{attribute addProperty Name "Pneumatic cyclinder"}
FUNCTION_BLOCK fbPiston EXTENDS TcoCore.TcoComponent IMPLEMENTS IPistonGripper, IPistonHorizontal, IPistonVertical
VAR_INPUT
	iHomePositionSensor : BOOL;
	iWorkPositionSensor : BOOL;	
END_VAR

VAR_OUTPUT
	qHomePositionActuator : BOOL;
	qWorkPositionActuator : BOOL;		
END_VAR

VAR
	{attribute addProperty Activity "moves to home position"}
	_moveHomeTask : fbPistonMoveTask(THIS^);
	{attribute addProperty Activity "moves to work position"}
	_moveWorkTask : fbPistonMoveTask(THIS^);
	_moveHomeMomentaryTask : TcoCore.TcoMomentaryTask(THIS^);	
	_moveHomeToggleTask : TcoCore.TcoToggleTask(THIS^, FALSE);
	
	_config : fbPistonConfig;
	_status : fbPistonStatus;
END_VAR

_moveHomeTask(PositionSensor := iHomePositionSensor, MoveToPositionSignal := qHomePositionActuator, InverseSignal := qWorkPositionActuator);
_moveWorkTask(PositionSensor := iWorkPositionSensor, MoveToPositionSignal := qWorkPositionActuator, InverseSignal := qHomePositionActuator);


_moveHomeMomentaryTask.Run();

_moveHomeToggleTask.Toggle();

METHOD Close : TcoCore.ITcoTaskStatus
Close := MoveToHome();
END_METHOD

METHOD MoveDown : TcoCore.ITcoTaskStatus
MoveDown := MoveToHome();
END_METHOD

METHOD MoveLeft : TcoCore.ITcoTaskStatus
MoveLeft := MoveToWork();
END_METHOD

METHOD MoveRight : TcoCore.ITcoTaskStatus
MoveRight := MoveToHome();
END_METHOD

METHOD PROTECTED MoveToHome : TcoCore.ITcoTaskStatus
MoveToHome := THIS^._moveHomeTask.Invoke();
END_METHOD

METHOD PROTECTED MoveToWork : TcoCore.ITcoTaskStatus
MoveToWork := THIS^._moveWorkTask.Invoke();
END_METHOD

METHOD MoveUp : TcoCore.ITcoTaskStatus
MoveUp := MoveToWork();
END_METHOD

METHOD Open : TcoCore.ITcoTaskStatus
Open := MoveToWork();
END_METHOD

METHOD  Restore : ITcoRestorable
THIS^._moveHomeTask.Restore();
THIS^._moveWorkTask.Restore();
END_METHOD

(*~
	<docu>
		<summary>
		    Custom service (manual, maintenance) logic.
			This method must be implemented in derived class.
		</summary>			
	</docu>	
~*)
METHOD PROTECTED  ServiceMode
END_METHOD

END_FUNCTION_BLOCK

(* stored: Version 1.1.0.1, ProductVersion 3.1.4024.9
   POU fbPiston: Id {3299369b-70c8-07a9-1d33-c5ca5f479567}, SpecialFunc None
   Folder Gripper: Id {7c77662b-e1b7-064c-3eef-f8b84e6fee58}
   Folder Horizontal: Id {a421e43c-bf24-02be-0068-4615a3275958}
   Folder Vertical: Id {c4d73989-33a4-024e-08c0-bd526bebe4e3}
   Method Close: Id {2a4f7cdc-5113-0359-390c-c200a7a27fa7}
   Method MoveDown: Id {9caa2779-f272-0a6e-0c4c-54a6dfa06add}
   Method MoveLeft: Id {8f619318-a724-0e44-3503-001490ed5b8c}
   Method MoveRight: Id {c80baeba-47e1-0722-3c87-e2f8baa67ff8}
   Method MoveToHome: Id {c882e135-b2d1-0271-100a-48513e6f381d}
   Method MoveToWork: Id {1d28b2df-661a-09ea-0d3b-89d31a065ff8}
   Method MoveUp: Id {f84f831b-d6b9-0bc0-3158-9924ccc80c44}
   Method Open: Id {07bb496f-8c19-03fc-3915-5004e4f348c2}
   Method Restore: Id {ce6d436c-62db-029a-3892-6da19ff128cd}
   Method ServiceMode: Id {3e528cd0-4ba9-0659-3710-db6acbc16678} *)
